TYPE "UDT_ZC_DISP_PPAL_EA"
VERSION : 0.1
   STRUCT
      ValorActual : Real;   // Valor actual
   END_STRUCT;

END_TYPE

